// TIA Portal V18 export
FUNCTION_BLOCK "auto_digital"   // FB12, FBD
{ S7_Optimized_Access := 'TRUE' }
VERSION : 0.1
// stored: AutoNumber true, IsIECCheckEnabled false, IsRetainMemResEnabled false, MemoryReserve 100, SetENOAutomatically false, UDAEnableTagReadback false
   VAR_INPUT
      ALLOWED : Bool;
      xFwdOK : Bool;
      xRevOK : Bool;
      xFwdFastOK : Bool;
      xRevFastOK : Bool;
   END_VAR
   VAR_OUTPUT
      FWD : Bool;
      REV : Bool;
      QUICK : Bool;
      status_fwd_full : Bool;
      status_mid : Bool;
      status_rev_full : Bool;
   END_VAR
   VAR_IN_OUT
      btn_go_fwd : Bool;
      btn_go_rev : Bool;
   END_VAR
   VAR
      lbs { S7_SetPoint := 'True'} : "last_button_stands";
      mem_fwdok : Bool;
      mem_revok : Bool;
      ton_quick { S7_SetPoint := 'True'} : TON_TIME;
   END_VAR
BEGIN

REGION Network 1
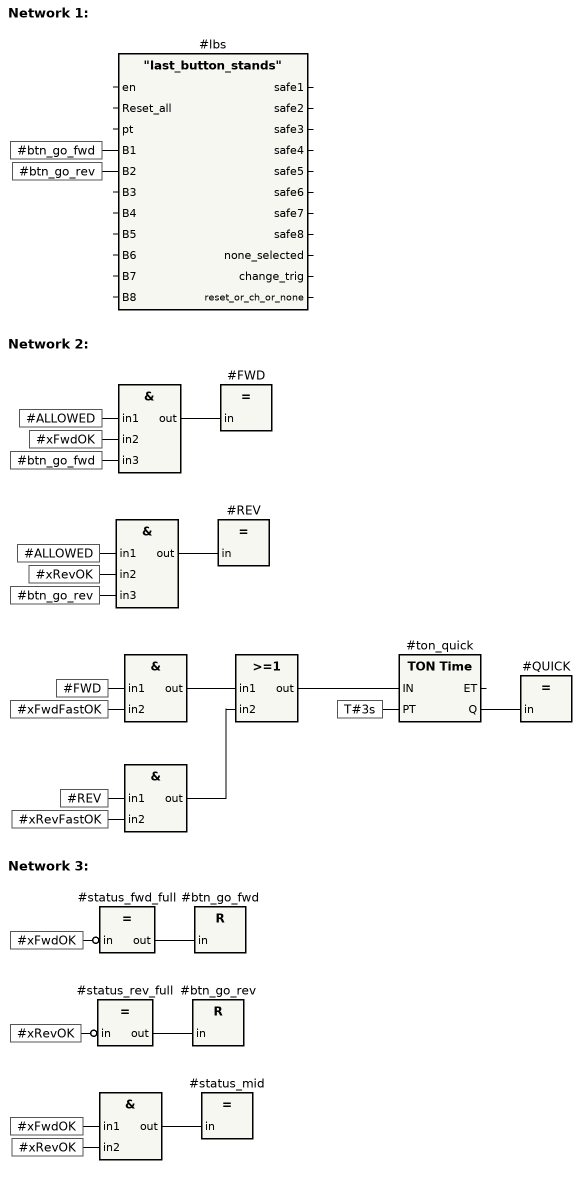
   #lbs(B1 := #btn_go_fwd, B2 := #btn_go_rev);   // "last_button_stands"
END_REGION

REGION Network 2
   #FWD := #ALLOWED AND #xFwdOK AND #btn_go_fwd;
   #REV := #ALLOWED AND #xRevOK AND #btn_go_rev;
   #ton_quick(IN := (#FWD AND #xFwdFastOK) OR (#REV AND #xRevFastOK), PT := T#3s);   // TON
   #QUICK := #ton_quick.Q;
END_REGION

REGION Network 3
   #status_fwd_full := NOT #xFwdOK;
   IF NOT #xFwdOK THEN #btn_go_fwd := FALSE; END_IF;
   #status_rev_full := NOT #xRevOK;
   IF NOT #xRevOK THEN #btn_go_rev := FALSE; END_IF;
   #status_mid := #xFwdOK AND #xRevOK;
END_REGION
END_FUNCTION_BLOCK
